// TIA Portal V17 export
// export: Created 2022-07-06T14:52:18.8349718Z, ExportSetting WithDefaults, DisplayName Totally Integrated Automation Portal, DisplayVersion V17 Update 4, DisplayName TIA Portal Openness, DisplayVersion V17 Update 4, DisplayName TIA Portal Version Control Interface, DisplayVersion V17, DisplayName STEP 7 Professional, DisplayVersion V17 Update 4, DisplayName STEP 7 CFC, DisplayVersion V17, DisplayName STEP 7 Safety, DisplayVersion V17, DisplayName WinCC Advanced, DisplayVersion V17 Update 4
FUNCTION_BLOCK "HMI_AB020_Fieldbus_02"   // FB69, FBD
{ S7_Optimized_Access := 'TRUE' }
VERSION : 0.1
// stored: AutoNumber true, IsIECCheckEnabled false, IsRetainMemResEnabled false, MemoryReserve 100, SetENOAutomatically false, UDAEnableTagReadback false
   VAR
      Message32_Flt100 { ExternalVisible := 'False'; ExternalWritable := 'False'; S7_SetPoint := 'True'} : "Message32";
      Message32_Flt2 { ExternalVisible := 'False'; ExternalWritable := 'False'; S7_SetPoint := 'True'} : "Message32";
      Message32_Flt3 { ExternalVisible := 'False'; ExternalWritable := 'False'; S7_SetPoint := 'True'} : "Message32";
      Message32_Flr4 { ExternalVisible := 'False'; ExternalWritable := 'False'; S7_SetPoint := 'True'} : "Message32";
      Message32_Wrn1 { ExternalVisible := 'False'; ExternalWritable := 'False'; S7_SetPoint := 'True'} : "Message32";
      Message32_Wrn2 { ExternalVisible := 'False'; ExternalWritable := 'False'; S7_SetPoint := 'True'} : "Message32";
      Message32_Wrn3 { ExternalVisible := 'False'; ExternalWritable := 'False'; S7_SetPoint := 'True'} : "Message32";
      Message32_Wrn4 { ExternalVisible := 'False'; ExternalWritable := 'False'; S7_SetPoint := 'True'} : "Message32";
   END_VAR
BEGIN

REGION Network 1: Not available slave 1-32
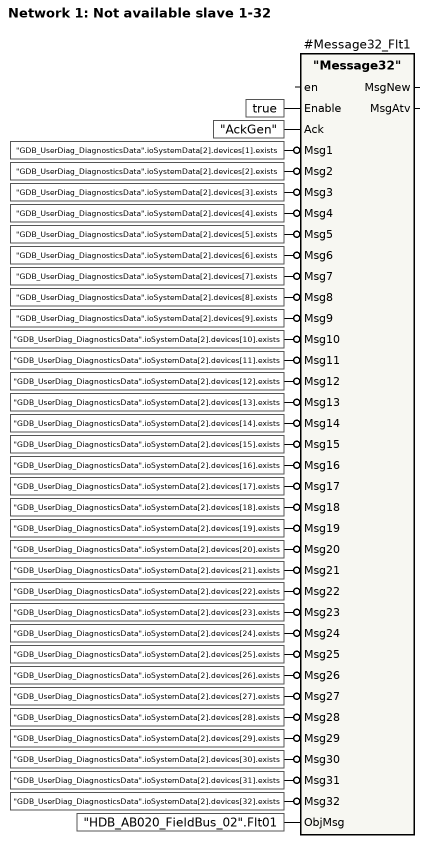
   #Message32_Flt1(Enable := true,   // "Message32"
                   Ack := "AckGen",
                   Msg1 := NOT "GDB_UserDiag_DiagnosticsData".ioSystemData[2].devices[1].exists,
                   Msg2 := NOT "GDB_UserDiag_DiagnosticsData".ioSystemData[2].devices[2].exists,
                   Msg3 := NOT "GDB_UserDiag_DiagnosticsData".ioSystemData[2].devices[3].exists,
                   Msg4 := NOT "GDB_UserDiag_DiagnosticsData".ioSystemData[2].devices[4].exists,
                   Msg5 := NOT "GDB_UserDiag_DiagnosticsData".ioSystemData[2].devices[5].exists,
                   Msg6 := NOT "GDB_UserDiag_DiagnosticsData".ioSystemData[2].devices[6].exists,
                   Msg7 := NOT "GDB_UserDiag_DiagnosticsData".ioSystemData[2].devices[7].exists,
                   Msg8 := NOT "GDB_UserDiag_DiagnosticsData".ioSystemData[2].devices[8].exists,
                   Msg9 := NOT "GDB_UserDiag_DiagnosticsData".ioSystemData[2].devices[9].exists,
                   Msg10 := NOT "GDB_UserDiag_DiagnosticsData".ioSystemData[2].devices[10].exists,
                   Msg11 := NOT "GDB_UserDiag_DiagnosticsData".ioSystemData[2].devices[11].exists,
                   Msg12 := NOT "GDB_UserDiag_DiagnosticsData".ioSystemData[2].devices[12].exists,
                   Msg13 := NOT "GDB_UserDiag_DiagnosticsData".ioSystemData[2].devices[13].exists,
                   Msg14 := NOT "GDB_UserDiag_DiagnosticsData".ioSystemData[2].devices[14].exists,
                   Msg15 := NOT "GDB_UserDiag_DiagnosticsData".ioSystemData[2].devices[15].exists,
                   Msg16 := NOT "GDB_UserDiag_DiagnosticsData".ioSystemData[2].devices[16].exists,
                   Msg17 := NOT "GDB_UserDiag_DiagnosticsData".ioSystemData[2].devices[17].exists,
                   Msg18 := NOT "GDB_UserDiag_DiagnosticsData".ioSystemData[2].devices[18].exists,
                   Msg19 := NOT "GDB_UserDiag_DiagnosticsData".ioSystemData[2].devices[19].exists,
                   Msg20 := NOT "GDB_UserDiag_DiagnosticsData".ioSystemData[2].devices[20].exists,
                   Msg21 := NOT "GDB_UserDiag_DiagnosticsData".ioSystemData[2].devices[21].exists,
                   Msg22 := NOT "GDB_UserDiag_DiagnosticsData".ioSystemData[2].devices[22].exists,
                   Msg23 := NOT "GDB_UserDiag_DiagnosticsData".ioSystemData[2].devices[23].exists,
                   Msg24 := NOT "GDB_UserDiag_DiagnosticsData".ioSystemData[2].devices[24].exists,
                   Msg25 := NOT "GDB_UserDiag_DiagnosticsData".ioSystemData[2].devices[25].exists,
                   Msg26 := NOT "GDB_UserDiag_DiagnosticsData".ioSystemData[2].devices[26].exists,
                   Msg27 := NOT "GDB_UserDiag_DiagnosticsData".ioSystemData[2].devices[27].exists,
                   Msg28 := NOT "GDB_UserDiag_DiagnosticsData".ioSystemData[2].devices[28].exists,
                   Msg29 := NOT "GDB_UserDiag_DiagnosticsData".ioSystemData[2].devices[29].exists,
                   Msg30 := NOT "GDB_UserDiag_DiagnosticsData".ioSystemData[2].devices[30].exists,
                   Msg31 := NOT "GDB_UserDiag_DiagnosticsData".ioSystemData[2].devices[31].exists,
                   Msg32 := NOT "GDB_UserDiag_DiagnosticsData".ioSystemData[2].devices[32].exists,
                   ObjMsg := "HDB_AB020_FieldBus_02".Flt01);
END_REGION

REGION Network 2: Not available slave 33-64
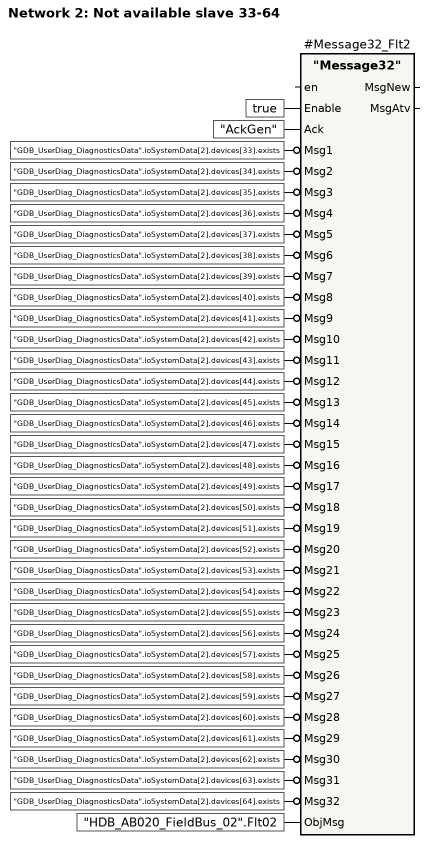
   #Message32_Flt2(Enable := true,   // "Message32"
                   Ack := "AckGen",
                   Msg1 := NOT "GDB_UserDiag_DiagnosticsData".ioSystemData[2].devices[33].exists,
                   Msg2 := NOT "GDB_UserDiag_DiagnosticsData".ioSystemData[2].devices[34].exists,
                   Msg3 := NOT "GDB_UserDiag_DiagnosticsData".ioSystemData[2].devices[35].exists,
                   Msg4 := NOT "GDB_UserDiag_DiagnosticsData".ioSystemData[2].devices[36].exists,
                   Msg5 := NOT "GDB_UserDiag_DiagnosticsData".ioSystemData[2].devices[37].exists,
                   Msg6 := NOT "GDB_UserDiag_DiagnosticsData".ioSystemData[2].devices[38].exists,
                   Msg7 := NOT "GDB_UserDiag_DiagnosticsData".ioSystemData[2].devices[39].exists,
                   Msg8 := NOT "GDB_UserDiag_DiagnosticsData".ioSystemData[2].devices[40].exists,
                   Msg9 := NOT "GDB_UserDiag_DiagnosticsData".ioSystemData[2].devices[41].exists,
                   Msg10 := NOT "GDB_UserDiag_DiagnosticsData".ioSystemData[2].devices[42].exists,
                   Msg11 := NOT "GDB_UserDiag_DiagnosticsData".ioSystemData[2].devices[43].exists,
                   Msg12 := NOT "GDB_UserDiag_DiagnosticsData".ioSystemData[2].devices[44].exists,
                   Msg13 := NOT "GDB_UserDiag_DiagnosticsData".ioSystemData[2].devices[45].exists,
                   Msg14 := NOT "GDB_UserDiag_DiagnosticsData".ioSystemData[2].devices[46].exists,
                   Msg15 := NOT "GDB_UserDiag_DiagnosticsData".ioSystemData[2].devices[47].exists,
                   Msg16 := NOT "GDB_UserDiag_DiagnosticsData".ioSystemData[2].devices[48].exists,
                   Msg17 := NOT "GDB_UserDiag_DiagnosticsData".ioSystemData[2].devices[49].exists,
                   Msg18 := NOT "GDB_UserDiag_DiagnosticsData".ioSystemData[2].devices[50].exists,
                   Msg19 := NOT "GDB_UserDiag_DiagnosticsData".ioSystemData[2].devices[51].exists,
                   Msg20 := NOT "GDB_UserDiag_DiagnosticsData".ioSystemData[2].devices[52].exists,
                   Msg21 := NOT "GDB_UserDiag_DiagnosticsData".ioSystemData[2].devices[53].exists,
                   Msg22 := NOT "GDB_UserDiag_DiagnosticsData".ioSystemData[2].devices[54].exists,
                   Msg23 := NOT "GDB_UserDiag_DiagnosticsData".ioSystemData[2].devices[55].exists,
                   Msg24 := NOT "GDB_UserDiag_DiagnosticsData".ioSystemData[2].devices[56].exists,
                   Msg25 := NOT "GDB_UserDiag_DiagnosticsData".ioSystemData[2].devices[57].exists,
                   Msg26 := NOT "GDB_UserDiag_DiagnosticsData".ioSystemData[2].devices[58].exists,
                   Msg27 := NOT "GDB_UserDiag_DiagnosticsData".ioSystemData[2].devices[59].exists,
                   Msg28 := NOT "GDB_UserDiag_DiagnosticsData".ioSystemData[2].devices[60].exists,
                   Msg29 := NOT "GDB_UserDiag_DiagnosticsData".ioSystemData[2].devices[61].exists,
                   Msg30 := NOT "GDB_UserDiag_DiagnosticsData".ioSystemData[2].devices[62].exists,
                   Msg31 := NOT "GDB_UserDiag_DiagnosticsData".ioSystemData[2].devices[63].exists,
                   Msg32 := NOT "GDB_UserDiag_DiagnosticsData".ioSystemData[2].devices[64].exists,
                   ObjMsg := "HDB_AB020_FieldBus_02".Flt02);
END_REGION

REGION Network 3: Not available slave 65-96
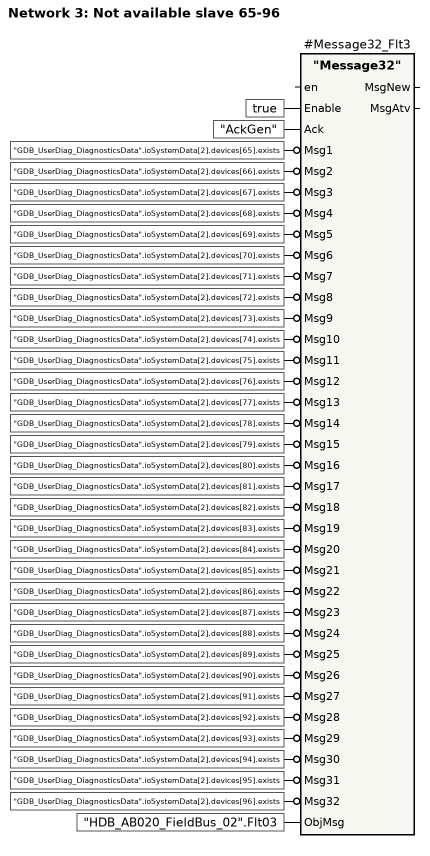
   #Message32_Flt3(Enable := true,   // "Message32"
                   Ack := "AckGen",
                   Msg1 := NOT "GDB_UserDiag_DiagnosticsData".ioSystemData[2].devices[65].exists,
                   Msg2 := NOT "GDB_UserDiag_DiagnosticsData".ioSystemData[2].devices[66].exists,
                   Msg3 := NOT "GDB_UserDiag_DiagnosticsData".ioSystemData[2].devices[67].exists,
                   Msg4 := NOT "GDB_UserDiag_DiagnosticsData".ioSystemData[2].devices[68].exists,
                   Msg5 := NOT "GDB_UserDiag_DiagnosticsData".ioSystemData[2].devices[69].exists,
                   Msg6 := NOT "GDB_UserDiag_DiagnosticsData".ioSystemData[2].devices[70].exists,
                   Msg7 := NOT "GDB_UserDiag_DiagnosticsData".ioSystemData[2].devices[71].exists,
                   Msg8 := NOT "GDB_UserDiag_DiagnosticsData".ioSystemData[2].devices[72].exists,
                   Msg9 := NOT "GDB_UserDiag_DiagnosticsData".ioSystemData[2].devices[73].exists,
                   Msg10 := NOT "GDB_UserDiag_DiagnosticsData".ioSystemData[2].devices[74].exists,
                   Msg11 := NOT "GDB_UserDiag_DiagnosticsData".ioSystemData[2].devices[75].exists,
                   Msg12 := NOT "GDB_UserDiag_DiagnosticsData".ioSystemData[2].devices[76].exists,
                   Msg13 := NOT "GDB_UserDiag_DiagnosticsData".ioSystemData[2].devices[77].exists,
                   Msg14 := NOT "GDB_UserDiag_DiagnosticsData".ioSystemData[2].devices[78].exists,
                   Msg15 := NOT "GDB_UserDiag_DiagnosticsData".ioSystemData[2].devices[79].exists,
                   Msg16 := NOT "GDB_UserDiag_DiagnosticsData".ioSystemData[2].devices[80].exists,
                   Msg17 := NOT "GDB_UserDiag_DiagnosticsData".ioSystemData[2].devices[81].exists,
                   Msg18 := NOT "GDB_UserDiag_DiagnosticsData".ioSystemData[2].devices[82].exists,
                   Msg19 := NOT "GDB_UserDiag_DiagnosticsData".ioSystemData[2].devices[83].exists,
                   Msg20 := NOT "GDB_UserDiag_DiagnosticsData".ioSystemData[2].devices[84].exists,
                   Msg21 := NOT "GDB_UserDiag_DiagnosticsData".ioSystemData[2].devices[85].exists,
                   Msg22 := NOT "GDB_UserDiag_DiagnosticsData".ioSystemData[2].devices[86].exists,
                   Msg23 := NOT "GDB_UserDiag_DiagnosticsData".ioSystemData[2].devices[87].exists,
                   Msg24 := NOT "GDB_UserDiag_DiagnosticsData".ioSystemData[2].devices[88].exists,
                   Msg25 := NOT "GDB_UserDiag_DiagnosticsData".ioSystemData[2].devices[89].exists,
                   Msg26 := NOT "GDB_UserDiag_DiagnosticsData".ioSystemData[2].devices[90].exists,
                   Msg27 := NOT "GDB_UserDiag_DiagnosticsData".ioSystemData[2].devices[91].exists,
                   Msg28 := NOT "GDB_UserDiag_DiagnosticsData".ioSystemData[2].devices[92].exists,
                   Msg29 := NOT "GDB_UserDiag_DiagnosticsData".ioSystemData[2].devices[93].exists,
                   Msg30 := NOT "GDB_UserDiag_DiagnosticsData".ioSystemData[2].devices[94].exists,
                   Msg31 := NOT "GDB_UserDiag_DiagnosticsData".ioSystemData[2].devices[95].exists,
                   Msg32 := NOT "GDB_UserDiag_DiagnosticsData".ioSystemData[2].devices[96].exists,
                   ObjMsg := "HDB_AB020_FieldBus_02".Flt03);
END_REGION

REGION Network 4: Not available slave 97-128
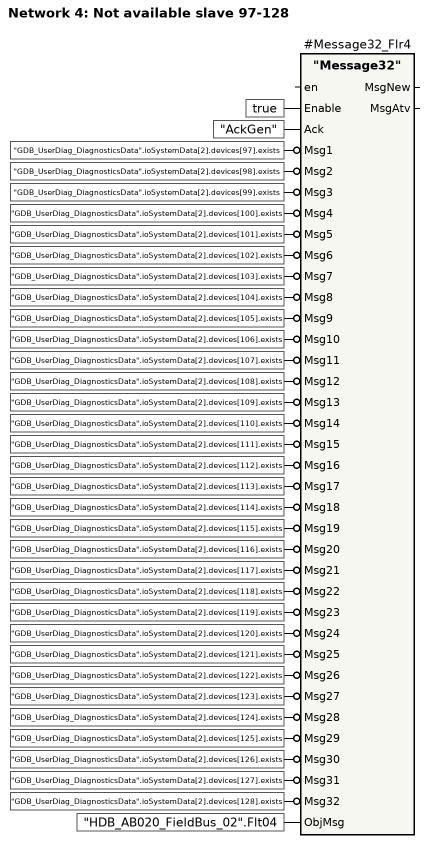
   #Message32_Flr4(Enable := true,   // "Message32"
                   Ack := "AckGen",
                   Msg1 := NOT "GDB_UserDiag_DiagnosticsData".ioSystemData[2].devices[97].exists,
                   Msg2 := NOT "GDB_UserDiag_DiagnosticsData".ioSystemData[2].devices[98].exists,
                   Msg3 := NOT "GDB_UserDiag_DiagnosticsData".ioSystemData[2].devices[99].exists,
                   Msg4 := NOT "GDB_UserDiag_DiagnosticsData".ioSystemData[2].devices[100].exists,
                   Msg5 := NOT "GDB_UserDiag_DiagnosticsData".ioSystemData[2].devices[101].exists,
                   Msg6 := NOT "GDB_UserDiag_DiagnosticsData".ioSystemData[2].devices[102].exists,
                   Msg7 := NOT "GDB_UserDiag_DiagnosticsData".ioSystemData[2].devices[103].exists,
                   Msg8 := NOT "GDB_UserDiag_DiagnosticsData".ioSystemData[2].devices[104].exists,
                   Msg9 := NOT "GDB_UserDiag_DiagnosticsData".ioSystemData[2].devices[105].exists,
                   Msg10 := NOT "GDB_UserDiag_DiagnosticsData".ioSystemData[2].devices[106].exists,
                   Msg11 := NOT "GDB_UserDiag_DiagnosticsData".ioSystemData[2].devices[107].exists,
                   Msg12 := NOT "GDB_UserDiag_DiagnosticsData".ioSystemData[2].devices[108].exists,
                   Msg13 := NOT "GDB_UserDiag_DiagnosticsData".ioSystemData[2].devices[109].exists,
                   Msg14 := NOT "GDB_UserDiag_DiagnosticsData".ioSystemData[2].devices[110].exists,
                   Msg15 := NOT "GDB_UserDiag_DiagnosticsData".ioSystemData[2].devices[111].exists,
                   Msg16 := NOT "GDB_UserDiag_DiagnosticsData".ioSystemData[2].devices[112].exists,
                   Msg17 := NOT "GDB_UserDiag_DiagnosticsData".ioSystemData[2].devices[113].exists,
                   Msg18 := NOT "GDB_UserDiag_DiagnosticsData".ioSystemData[2].devices[114].exists,
                   Msg19 := NOT "GDB_UserDiag_DiagnosticsData".ioSystemData[2].devices[115].exists,
                   Msg20 := NOT "GDB_UserDiag_DiagnosticsData".ioSystemData[2].devices[116].exists,
                   Msg21 := NOT "GDB_UserDiag_DiagnosticsData".ioSystemData[2].devices[117].exists,
                   Msg22 := NOT "GDB_UserDiag_DiagnosticsData".ioSystemData[2].devices[118].exists,
                   Msg23 := NOT "GDB_UserDiag_DiagnosticsData".ioSystemData[2].devices[119].exists,
                   Msg24 := NOT "GDB_UserDiag_DiagnosticsData".ioSystemData[2].devices[120].exists,
                   Msg25 := NOT "GDB_UserDiag_DiagnosticsData".ioSystemData[2].devices[121].exists,
                   Msg26 := NOT "GDB_UserDiag_DiagnosticsData".ioSystemData[2].devices[122].exists,
                   Msg27 := NOT "GDB_UserDiag_DiagnosticsData".ioSystemData[2].devices[123].exists,
                   Msg28 := NOT "GDB_UserDiag_DiagnosticsData".ioSystemData[2].devices[124].exists,
                   Msg29 := NOT "GDB_UserDiag_DiagnosticsData".ioSystemData[2].devices[125].exists,
                   Msg30 := NOT "GDB_UserDiag_DiagnosticsData".ioSystemData[2].devices[126].exists,
                   Msg31 := NOT "GDB_UserDiag_DiagnosticsData".ioSystemData[2].devices[127].exists,
                   Msg32 := NOT "GDB_UserDiag_DiagnosticsData".ioSystemData[2].devices[128].exists,
                   ObjMsg := "HDB_AB020_FieldBus_02".Flt04);
END_REGION

REGION Network 5: Problem Slave 1-32
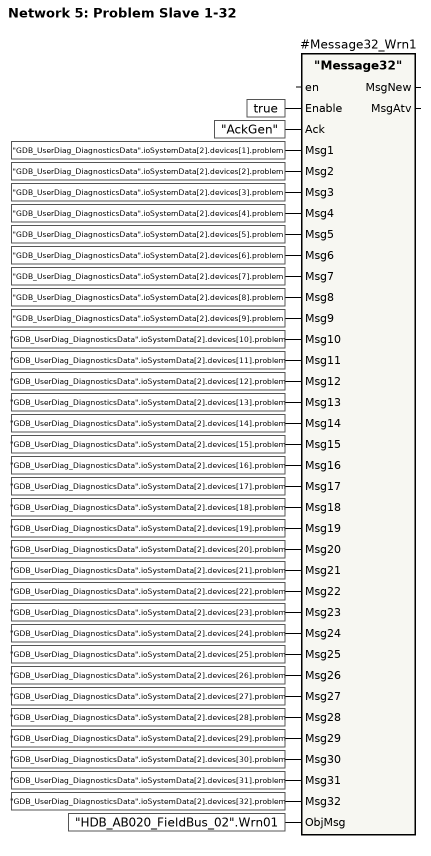
   #Message32_Wrn1(Enable := true,   // "Message32"
                   Ack := "AckGen",
                   Msg1 := "GDB_UserDiag_DiagnosticsData".ioSystemData[2].devices[1].problem,
                   Msg2 := "GDB_UserDiag_DiagnosticsData".ioSystemData[2].devices[2].problem,
                   Msg3 := "GDB_UserDiag_DiagnosticsData".ioSystemData[2].devices[3].problem,
                   Msg4 := "GDB_UserDiag_DiagnosticsData".ioSystemData[2].devices[4].problem,
                   Msg5 := "GDB_UserDiag_DiagnosticsData".ioSystemData[2].devices[5].problem,
                   Msg6 := "GDB_UserDiag_DiagnosticsData".ioSystemData[2].devices[6].problem,
                   Msg7 := "GDB_UserDiag_DiagnosticsData".ioSystemData[2].devices[7].problem,
                   Msg8 := "GDB_UserDiag_DiagnosticsData".ioSystemData[2].devices[8].problem,
                   Msg9 := "GDB_UserDiag_DiagnosticsData".ioSystemData[2].devices[9].problem,
                   Msg10 := "GDB_UserDiag_DiagnosticsData".ioSystemData[2].devices[10].problem,
                   Msg11 := "GDB_UserDiag_DiagnosticsData".ioSystemData[2].devices[11].problem,
                   Msg12 := "GDB_UserDiag_DiagnosticsData".ioSystemData[2].devices[12].problem,
                   Msg13 := "GDB_UserDiag_DiagnosticsData".ioSystemData[2].devices[13].problem,
                   Msg14 := "GDB_UserDiag_DiagnosticsData".ioSystemData[2].devices[14].problem,
                   Msg15 := "GDB_UserDiag_DiagnosticsData".ioSystemData[2].devices[15].problem,
                   Msg16 := "GDB_UserDiag_DiagnosticsData".ioSystemData[2].devices[16].problem,
                   Msg17 := "GDB_UserDiag_DiagnosticsData".ioSystemData[2].devices[17].problem,
                   Msg18 := "GDB_UserDiag_DiagnosticsData".ioSystemData[2].devices[18].problem,
                   Msg19 := "GDB_UserDiag_DiagnosticsData".ioSystemData[2].devices[19].problem,
                   Msg20 := "GDB_UserDiag_DiagnosticsData".ioSystemData[2].devices[20].problem,
                   Msg21 := "GDB_UserDiag_DiagnosticsData".ioSystemData[2].devices[21].problem,
                   Msg22 := "GDB_UserDiag_DiagnosticsData".ioSystemData[2].devices[22].problem,
                   Msg23 := "GDB_UserDiag_DiagnosticsData".ioSystemData[2].devices[23].problem,
                   Msg24 := "GDB_UserDiag_DiagnosticsData".ioSystemData[2].devices[24].problem,
                   Msg25 := "GDB_UserDiag_DiagnosticsData".ioSystemData[2].devices[25].problem,
                   Msg26 := "GDB_UserDiag_DiagnosticsData".ioSystemData[2].devices[26].problem,
                   Msg27 := "GDB_UserDiag_DiagnosticsData".ioSystemData[2].devices[27].problem,
                   Msg28 := "GDB_UserDiag_DiagnosticsData".ioSystemData[2].devices[28].problem,
                   Msg29 := "GDB_UserDiag_DiagnosticsData".ioSystemData[2].devices[29].problem,
                   Msg30 := "GDB_UserDiag_DiagnosticsData".ioSystemData[2].devices[30].problem,
                   Msg31 := "GDB_UserDiag_DiagnosticsData".ioSystemData[2].devices[31].problem,
                   Msg32 := "GDB_UserDiag_DiagnosticsData".ioSystemData[2].devices[32].problem,
                   ObjMsg := "HDB_AB020_FieldBus_02".Wrn01);
END_REGION

REGION Network 6: Problem Slave 33-64
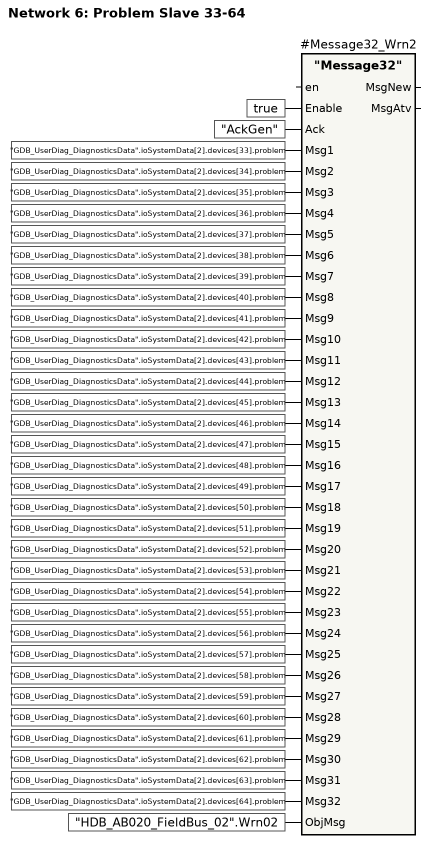
   #Message32_Wrn2(Enable := true,   // "Message32"
                   Ack := "AckGen",
                   Msg1 := "GDB_UserDiag_DiagnosticsData".ioSystemData[2].devices[33].problem,
                   Msg2 := "GDB_UserDiag_DiagnosticsData".ioSystemData[2].devices[34].problem,
                   Msg3 := "GDB_UserDiag_DiagnosticsData".ioSystemData[2].devices[35].problem,
                   Msg4 := "GDB_UserDiag_DiagnosticsData".ioSystemData[2].devices[36].problem,
                   Msg5 := "GDB_UserDiag_DiagnosticsData".ioSystemData[2].devices[37].problem,
                   Msg6 := "GDB_UserDiag_DiagnosticsData".ioSystemData[2].devices[38].problem,
                   Msg7 := "GDB_UserDiag_DiagnosticsData".ioSystemData[2].devices[39].problem,
                   Msg8 := "GDB_UserDiag_DiagnosticsData".ioSystemData[2].devices[40].problem,
                   Msg9 := "GDB_UserDiag_DiagnosticsData".ioSystemData[2].devices[41].problem,
                   Msg10 := "GDB_UserDiag_DiagnosticsData".ioSystemData[2].devices[42].problem,
                   Msg11 := "GDB_UserDiag_DiagnosticsData".ioSystemData[2].devices[43].problem,
                   Msg12 := "GDB_UserDiag_DiagnosticsData".ioSystemData[2].devices[44].problem,
                   Msg13 := "GDB_UserDiag_DiagnosticsData".ioSystemData[2].devices[45].problem,
                   Msg14 := "GDB_UserDiag_DiagnosticsData".ioSystemData[2].devices[46].problem,
                   Msg15 := "GDB_UserDiag_DiagnosticsData".ioSystemData[2].devices[47].problem,
                   Msg16 := "GDB_UserDiag_DiagnosticsData".ioSystemData[2].devices[48].problem,
                   Msg17 := "GDB_UserDiag_DiagnosticsData".ioSystemData[2].devices[49].problem,
                   Msg18 := "GDB_UserDiag_DiagnosticsData".ioSystemData[2].devices[50].problem,
                   Msg19 := "GDB_UserDiag_DiagnosticsData".ioSystemData[2].devices[51].problem,
                   Msg20 := "GDB_UserDiag_DiagnosticsData".ioSystemData[2].devices[52].problem,
                   Msg21 := "GDB_UserDiag_DiagnosticsData".ioSystemData[2].devices[53].problem,
                   Msg22 := "GDB_UserDiag_DiagnosticsData".ioSystemData[2].devices[54].problem,
                   Msg23 := "GDB_UserDiag_DiagnosticsData".ioSystemData[2].devices[55].problem,
                   Msg24 := "GDB_UserDiag_DiagnosticsData".ioSystemData[2].devices[56].problem,
                   Msg25 := "GDB_UserDiag_DiagnosticsData".ioSystemData[2].devices[57].problem,
                   Msg26 := "GDB_UserDiag_DiagnosticsData".ioSystemData[2].devices[58].problem,
                   Msg27 := "GDB_UserDiag_DiagnosticsData".ioSystemData[2].devices[59].problem,
                   Msg28 := "GDB_UserDiag_DiagnosticsData".ioSystemData[2].devices[60].problem,
                   Msg29 := "GDB_UserDiag_DiagnosticsData".ioSystemData[2].devices[61].problem,
                   Msg30 := "GDB_UserDiag_DiagnosticsData".ioSystemData[2].devices[62].problem,
                   Msg31 := "GDB_UserDiag_DiagnosticsData".ioSystemData[2].devices[63].problem,
                   Msg32 := "GDB_UserDiag_DiagnosticsData".ioSystemData[2].devices[64].problem,
                   ObjMsg := "HDB_AB020_FieldBus_02".Wrn02);
END_REGION

REGION Network 7: Problem Slave 65-96
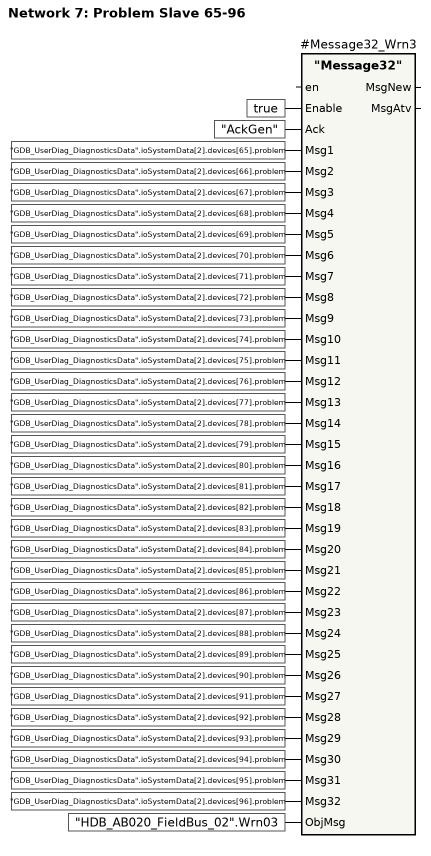
   #Message32_Wrn3(Enable := true,   // "Message32"
                   Ack := "AckGen",
                   Msg1 := "GDB_UserDiag_DiagnosticsData".ioSystemData[2].devices[65].problem,
                   Msg2 := "GDB_UserDiag_DiagnosticsData".ioSystemData[2].devices[66].problem,
                   Msg3 := "GDB_UserDiag_DiagnosticsData".ioSystemData[2].devices[67].problem,
                   Msg4 := "GDB_UserDiag_DiagnosticsData".ioSystemData[2].devices[68].problem,
                   Msg5 := "GDB_UserDiag_DiagnosticsData".ioSystemData[2].devices[69].problem,
                   Msg6 := "GDB_UserDiag_DiagnosticsData".ioSystemData[2].devices[70].problem,
                   Msg7 := "GDB_UserDiag_DiagnosticsData".ioSystemData[2].devices[71].problem,
                   Msg8 := "GDB_UserDiag_DiagnosticsData".ioSystemData[2].devices[72].problem,
                   Msg9 := "GDB_UserDiag_DiagnosticsData".ioSystemData[2].devices[73].problem,
                   Msg10 := "GDB_UserDiag_DiagnosticsData".ioSystemData[2].devices[74].problem,
                   Msg11 := "GDB_UserDiag_DiagnosticsData".ioSystemData[2].devices[75].problem,
                   Msg12 := "GDB_UserDiag_DiagnosticsData".ioSystemData[2].devices[76].problem,
                   Msg13 := "GDB_UserDiag_DiagnosticsData".ioSystemData[2].devices[77].problem,
                   Msg14 := "GDB_UserDiag_DiagnosticsData".ioSystemData[2].devices[78].problem,
                   Msg15 := "GDB_UserDiag_DiagnosticsData".ioSystemData[2].devices[79].problem,
                   Msg16 := "GDB_UserDiag_DiagnosticsData".ioSystemData[2].devices[80].problem,
                   Msg17 := "GDB_UserDiag_DiagnosticsData".ioSystemData[2].devices[81].problem,
                   Msg18 := "GDB_UserDiag_DiagnosticsData".ioSystemData[2].devices[82].problem,
                   Msg19 := "GDB_UserDiag_DiagnosticsData".ioSystemData[2].devices[83].problem,
                   Msg20 := "GDB_UserDiag_DiagnosticsData".ioSystemData[2].devices[84].problem,
                   Msg21 := "GDB_UserDiag_DiagnosticsData".ioSystemData[2].devices[85].problem,
                   Msg22 := "GDB_UserDiag_DiagnosticsData".ioSystemData[2].devices[86].problem,
                   Msg23 := "GDB_UserDiag_DiagnosticsData".ioSystemData[2].devices[87].problem,
                   Msg24 := "GDB_UserDiag_DiagnosticsData".ioSystemData[2].devices[88].problem,
                   Msg25 := "GDB_UserDiag_DiagnosticsData".ioSystemData[2].devices[89].problem,
                   Msg26 := "GDB_UserDiag_DiagnosticsData".ioSystemData[2].devices[90].problem,
                   Msg27 := "GDB_UserDiag_DiagnosticsData".ioSystemData[2].devices[91].problem,
                   Msg28 := "GDB_UserDiag_DiagnosticsData".ioSystemData[2].devices[92].problem,
                   Msg29 := "GDB_UserDiag_DiagnosticsData".ioSystemData[2].devices[93].problem,
                   Msg30 := "GDB_UserDiag_DiagnosticsData".ioSystemData[2].devices[94].problem,
                   Msg31 := "GDB_UserDiag_DiagnosticsData".ioSystemData[2].devices[95].problem,
                   Msg32 := "GDB_UserDiag_DiagnosticsData".ioSystemData[2].devices[96].problem,
                   ObjMsg := "HDB_AB020_FieldBus_02".Wrn03);
END_REGION

REGION Network 8: Problem Slave 97-128
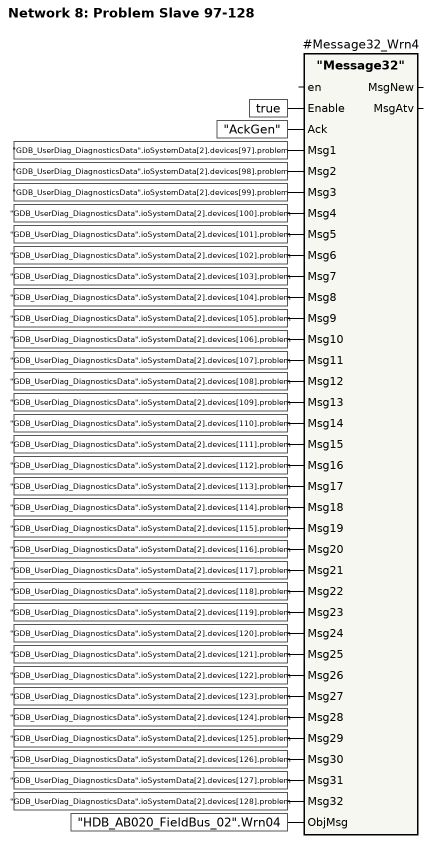
   #Message32_Wrn4(Enable := true,   // "Message32"
                   Ack := "AckGen",
                   Msg1 := "GDB_UserDiag_DiagnosticsData".ioSystemData[2].devices[97].problem,
                   Msg2 := "GDB_UserDiag_DiagnosticsData".ioSystemData[2].devices[98].problem,
                   Msg3 := "GDB_UserDiag_DiagnosticsData".ioSystemData[2].devices[99].problem,
                   Msg4 := "GDB_UserDiag_DiagnosticsData".ioSystemData[2].devices[100].problem,
                   Msg5 := "GDB_UserDiag_DiagnosticsData".ioSystemData[2].devices[101].problem,
                   Msg6 := "GDB_UserDiag_DiagnosticsData".ioSystemData[2].devices[102].problem,
                   Msg7 := "GDB_UserDiag_DiagnosticsData".ioSystemData[2].devices[103].problem,
                   Msg8 := "GDB_UserDiag_DiagnosticsData".ioSystemData[2].devices[104].problem,
                   Msg9 := "GDB_UserDiag_DiagnosticsData".ioSystemData[2].devices[105].problem,
                   Msg10 := "GDB_UserDiag_DiagnosticsData".ioSystemData[2].devices[106].problem,
                   Msg11 := "GDB_UserDiag_DiagnosticsData".ioSystemData[2].devices[107].problem,
                   Msg12 := "GDB_UserDiag_DiagnosticsData".ioSystemData[2].devices[108].problem,
                   Msg13 := "GDB_UserDiag_DiagnosticsData".ioSystemData[2].devices[109].problem,
                   Msg14 := "GDB_UserDiag_DiagnosticsData".ioSystemData[2].devices[110].problem,
                   Msg15 := "GDB_UserDiag_DiagnosticsData".ioSystemData[2].devices[111].problem,
                   Msg16 := "GDB_UserDiag_DiagnosticsData".ioSystemData[2].devices[112].problem,
                   Msg17 := "GDB_UserDiag_DiagnosticsData".ioSystemData[2].devices[113].problem,
                   Msg18 := "GDB_UserDiag_DiagnosticsData".ioSystemData[2].devices[114].problem,
                   Msg19 := "GDB_UserDiag_DiagnosticsData".ioSystemData[2].devices[115].problem,
                   Msg20 := "GDB_UserDiag_DiagnosticsData".ioSystemData[2].devices[116].problem,
                   Msg21 := "GDB_UserDiag_DiagnosticsData".ioSystemData[2].devices[117].problem,
                   Msg22 := "GDB_UserDiag_DiagnosticsData".ioSystemData[2].devices[118].problem,
                   Msg23 := "GDB_UserDiag_DiagnosticsData".ioSystemData[2].devices[119].problem,
                   Msg24 := "GDB_UserDiag_DiagnosticsData".ioSystemData[2].devices[120].problem,
                   Msg25 := "GDB_UserDiag_DiagnosticsData".ioSystemData[2].devices[121].problem,
                   Msg26 := "GDB_UserDiag_DiagnosticsData".ioSystemData[2].devices[122].problem,
                   Msg27 := "GDB_UserDiag_DiagnosticsData".ioSystemData[2].devices[123].problem,
                   Msg28 := "GDB_UserDiag_DiagnosticsData".ioSystemData[2].devices[124].problem,
                   Msg29 := "GDB_UserDiag_DiagnosticsData".ioSystemData[2].devices[125].problem,
                   Msg30 := "GDB_UserDiag_DiagnosticsData".ioSystemData[2].devices[126].problem,
                   Msg31 := "GDB_UserDiag_DiagnosticsData".ioSystemData[2].devices[127].problem,
                   Msg32 := "GDB_UserDiag_DiagnosticsData".ioSystemData[2].devices[128].problem,
                   ObjMsg := "HDB_AB020_FieldBus_02".Wrn04);
END_REGION
END_FUNCTION_BLOCK
